(* PLC project BlogProject.project, CODESYS CODESYS V3.5 SP14 Patch 3 *)
(* stored: creationDateTime 2021-10-07T21:04:54.9241535, modificationDateTime 2021-10-07T20:40:20.1109198 *)

FUNCTION_BLOCK mcIsErrorReset IMPLEMENTS itfEvent
  VAR
    bErrorReset : BOOL;
  END_VAR

            
          

METHOD getEvent : BOOL
                  getEvent:=bErrorReset;
                
END_METHOD
END_FUNCTION_BLOCK
